(* CODESYS project PLS3 Flomsikring 28.07.2021.export

Project tree, tasks and I/O mapping:
  application PLS3_Flomsikring
    task MQTT (cyclic, interval 5000 ms, priority 15, watchdog 4500 ms x 1) calls Simulation_MQTT
    task PLC_Task (cyclic, interval 500 ms, priority 15, watchdog 400 ms x 1) calls PLC_PRG
    task VISU_TASK (cyclic, interval 100 ms, priority 15) calls VisuElems.Visu_Prg
    GlobalData/
      global variables HMI
      global variables IO
      global variables Local
      global variables SIM
      global variables STATUS
    LibFB/
      function block AlarmDigitalFB [ST]
      function block ControlAnalogFB [ST]
      function block MotorDigitalFB [ST]
      function block PIDFB [ST]
      function block PowerMonitoringFb [ST]
      function block ScalingFB [ST]
      function block SignalAnalogFB [ST]
      function block signalDigitalFB [ST]
      function block TimerFB [ST]
      function block WorkDistributorFB [ST]
    LibHmiStructs/
      data type AlarmDigitalHmiCmd
      data type AlarmDigitalHmiPv
      data type AliveHmiPv
      data type ControlAnalogHmiCmd
      data type ControlAnalogHmiPv
      data type MotorDigitalHmiCmd
      data type MotorDigitalHmiPv
      data type PIDHmiCmd
      data type PIDHmiPv
      data type PowerMonitoringHmiCmd
      data type PowerMonitoringHmiPv
      data type ScalingHmiCmd
      data type ScalingHmiPv
      data type SignalAnalogHmiCmd
      data type SignalAnalogHmiPv
      data type SignalDigitalHmiCmd
      data type SignalDigitalHmiPv
      data type TimerHmiCmd
      data type TimerHmiPv
      data type WorkDistributorHmiPv
    Utils/
      data type OpcUa_Mqtt_Status
      function eulers [ST]
      function firstOrderSystem [ST]
      function process [ST]
      function String_To_ForcastArray [ST]
    program Alarms [ST]
    program Control [ST]
    program Initialize [ST]
    program Inputs [ST]
    program Outputs [ST]
    program PLC_PRG [ST]
    function RestartOpcUaMqttLinkOnDownload [ST]
    function RestartOpcUaMqttLinkOnOnlineChange [ST]
    program Simulation [ST]
    program Simulation_MQTT [ST]
    global variables PersistentVars
    visualisation Visualization
*)

// PLS3_Flomsikring/LibHmiStructs/AlarmDigitalHmiCmd
// These are autogenerated, do not manual modify it
TYPE AlarmDigitalHmiCmd :
STRUCT
	_tagId: STRING;
	_type: STRING;
	_owner: STRING;
	Tag:	STRING;
	Description:	STRING;
	Delay:	TimerHmiCmd;
	Acknowledged:	BOOL;
END_STRUCT
END_TYPE

// PLS3_Flomsikring/LibHmiStructs/AlarmDigitalHmiPv
// These are autogenerated, do not manual modify it
TYPE AlarmDigitalHmiPv :
STRUCT
	_tagId: STRING;
	_type: STRING;
	_owner: STRING;
	Input_Pv:	BOOL;
	Delay:	TimerHmiPv;
	Alarm:	BOOL;
END_STRUCT
END_TYPE

// PLS3_Flomsikring/LibHmiStructs/AliveHmiPv
// These are autogenerated, do not manual modify it
TYPE AliveHmiPv :
STRUCT
	_tagId:STRING;
	_type: STRING;
	_owner: STRING;
	CounterPv:INT;
END_STRUCT
END_TYPE

// PLS3_Flomsikring/LibHmiStructs/ControlAnalogHmiCmd
// These are autogenerated, do not manual modify it
TYPE ControlAnalogHmiCmd :
STRUCT
	_tagId: STRING;
	_type: STRING;
	_owner: STRING;
	Tag:STRING;
	Description:STRING;
	Auto:BOOL;
	ManualControlValue_Cmd:REAL;
	AlarmControlFailed:	AlarmDigitalHmiCmd;
	AlarmControlFailedLimit:	REAL;
END_STRUCT
END_TYPE

// PLS3_Flomsikring/LibHmiStructs/ControlAnalogHmiPv
// These are autogenerated, do not manual modify it
TYPE ControlAnalogHmiPv :
STRUCT
	_tagId: STRING;
	_type: STRING;
	_owner: STRING;
	ControlValue_Pv:	REAL;
	Interlocked_Pv:	BOOL;
	AlarmControlFailed:	AlarmDigitalHmiPv;
	Feedback_Pv:REAL;
	RunHours_Pv:INT;
	RunMinutes_Pv:int;
END_STRUCT
END_TYPE

// PLS3_Flomsikring/LibHmiStructs/MotorDigitalHmiCmd
// These are autogenerated, do not manual modify it
TYPE MotorDigitalHmiCmd :
STRUCT
_tagId: STRING;
_type: STRING;
_owner: STRING;
Tag:STRING;
Description:STRING;
Auto:BOOL;
AlarmStartFailed:AlarmDigitalHmiCmd;
AlarmStopFailed:AlarmDigitalHmiCmd;
ManualStart_Cmd:BOOL;
END_STRUCT
END_TYPE

// PLS3_Flomsikring/LibHmiStructs/MotorDigitalHmiPv
// These are autogenerated, do not manual modify it
TYPE MotorDigitalHmiPv :
STRUCT
_tagId: STRING;
_type: STRING;
_owner: STRING;
Interlocked_Pv:BOOL;
ControlValue_Pv:BOOL;
AlarmStartFailed:AlarmDigitalHmiPv;
AlarmStopFailed:AlarmDigitalHmiPv;
Started_Pv:BOOL;
Stopped_Pv:BOOL;
END_STRUCT
END_TYPE

// PLS3_Flomsikring/LibHmiStructs/PIDHmiCmd
// These are autogenerated, do not manual modify it
TYPE PIDHmiCmd :
STRUCT
	_tagId: STRING;
	_type: STRING;
	_owner: STRING;
	Tag:STRING;
	Description:STRING;
	K:REAL;
	EnableK:BOOL;
	Ti:REAL;
	EnableI:BOOL;
	Td:REAL;
	N:REAL;
	EnableD:BOOL;
	Auto:BOOL;
	ManualValue_Cmd:REAL;
	u0:REAL;
	TrackingGain:REAL;
	HmiReference_Cmd:REAL;
	HmiReference:BOOL;
END_STRUCT
END_TYPE

// PLS3_Flomsikring/LibHmiStructs/PIDHmiPv
// These are autogenerated, do not manual modify it
TYPE PIDHmiPv :
STRUCT
	_tagId: STRING;
	_type: STRING;
	_owner: STRING;
	Reference_Pv:REAL;
	ProcessMeasure:REAL;
	Error:REAL;
	Output:REAL;
	up:REAL;
	ui:REAL;
	ud:REAL;
	es:REAL;
	u:REAL;
END_STRUCT
END_TYPE

// PLS3_Flomsikring/LibHmiStructs/PowerMonitoringHmiCmd
//These are autogenerated, do not manual modify it
TYPE PowerMonitoringHmiCmd :
STRUCT
	_tagId: STRING;
	_type: STRING;
	_owner: STRING;
	BatterySize_Cmd:REAL; //Size of the battery in mAh
END_STRUCT
END_TYPE

// PLS3_Flomsikring/LibHmiStructs/PowerMonitoringHmiPv
//These are autogenerated, do not manual modify it
TYPE PowerMonitoringHmiPv :
STRUCT
_tagId: STRING;
_type: STRING;
_owner: STRING;
Status_string:STRING;
Status_bool:BOOL;
Time_string:STRING;
Time_pv:REAL;
Alarm:BOOL;
Input_Current_In:REAL;
Input_Current_Out:REAL;
Input_Battery_Level:REAL;
END_STRUCT
END_TYPE

// PLS3_Flomsikring/LibHmiStructs/ScalingHmiCmd
// These are autogenerated, do not manual modify it
TYPE ScalingHmiCmd :
STRUCT
	_tagId: STRING;
	_type: STRING;
	_owner: STRING;
	InputUnit:STRING;
	InputMin_Cmd:REAL;
	InputMax_Cmd:REAL;
	OutputUnit:STRING;
	OutputMin_Cmd:REAL;
	OutputMax_Cmd:REAL;
END_STRUCT
END_TYPE

// PLS3_Flomsikring/LibHmiStructs/ScalingHmiPv
// These are autogenerated, do not manual modify it
TYPE ScalingHmiPv :
STRUCT
_tagId: STRING;
_type: STRING;
_owner: STRING;
Input_Pv:REAL;
Output_Pv:REAL;
END_STRUCT
END_TYPE

// PLS3_Flomsikring/LibHmiStructs/SignalAnalogHmiCmd
// These are autogenerated, do not manual modify it
TYPE SignalAnalogHmiCmd :
STRUCT
_tagId: STRING;
_type: STRING;
_owner: STRING;
Tag:STRING;
Description:STRING;
AlarmHigh:AlarmDigitalHmiCmd;
AlarmHighHigh:AlarmDigitalHmiCmd;
AlarmLow:AlarmDigitalHmiCmd;
AlarmLowLow:AlarmDigitalHmiCmd;
AlarmHighLimit:REAL;
AlarmHighHighLimit:REAL;
AlarmLowLimit:REAL;
AlarmLowLowLimit:REAL;
AlarmHysteresis:REAL;
SimulationMode:BOOL;
SimulationValue:REAL;
InputScaling:ScalingHmiCmd;
END_STRUCT
END_TYPE

// PLS3_Flomsikring/LibHmiStructs/SignalAnalogHmiPv
// These are autogenerated, do not manual modify it
TYPE SignalAnalogHmiPv :
STRUCT
_tagId: STRING;
_type: STRING;
_owner: STRING;
RawInput_Pv:REAL;
Output_Pv:REAL;
AlarmHigh:AlarmDigitalHmiPv;
AlarmHighHigh:AlarmDigitalHmiPv;
AlarmLow:AlarmDigitalHmiPv;
AlarmLowLow:AlarmDigitalHmiPv;
InputScaling:ScalingHmiPv;
END_STRUCT
END_TYPE

// PLS3_Flomsikring/LibHmiStructs/SignalDigitalHmiCmd
// These are autogenerated, do not manual modify it
TYPE SignalDigitalHmiCmd :
STRUCT
_tagId: STRING;
_type: STRING;
_owner: STRING;
Tag:STRING;
Description:STRING;
SimulationMode:BOOL;
SimulationValue:BOOL;
END_STRUCT
END_TYPE

// PLS3_Flomsikring/LibHmiStructs/SignalDigitalHmiPv
// These are autogenerated, do not manual modify it
TYPE SignalDigitalHmiPv :
STRUCT
_tagId: STRING;
_type: STRING;
_owner: STRING;
Input_Pv:BOOL;
Output_Pv:BOOL;
END_STRUCT
END_TYPE

// PLS3_Flomsikring/LibHmiStructs/TimerHmiCmd
// These are autogenerated, do not manual modify it
TYPE TimerHmiCmd :
STRUCT
	_tagId:STRING;
	_type: STRING;
	_owner: STRING;
	Tag:	STRING;
	Description:	STRING;
	OnDelayLimit:	REAL;
	OffDelayLimit:	REAL;
END_STRUCT
END_TYPE

// PLS3_Flomsikring/LibHmiStructs/TimerHmiPv
// These are autogenerated, do not manual modify it
TYPE TimerHmiPv :
STRUCT
	_tagId:STRING;
	_type: STRING;
	_owner: STRING;
	Input_Pv:	BOOL;
	Output_Pv:	BOOL;
	OnDelayElapsed:	REAL;
	OffDelayElapsed:	REAL;
END_STRUCT
END_TYPE

// PLS3_Flomsikring/LibHmiStructs/WorkDistributorHmiPv
// These are autogenerated, do not manual modify it
TYPE WorkDistributorHmiPv :
STRUCT
_tagId:STRING;
_type:STRING;
_owner:STRING;
Tag1:STRING;
Tag2:STRING;
Tag3:STRING;
RunHours1:INT;
RunHours2:INT;
RunHours3:INT;
AlarmNotAuto:BOOL;
END_STRUCT
END_TYPE

// PLS3_Flomsikring/Utils/OpcUa_Mqtt_Status
TYPE OpcUa_Mqtt_Status :
STRUCT
	LastRun:STRING;
	AliveCounterPv:INT := 0;
	Restart_Cmd:BOOL := FALSE;
END_STRUCT
END_TYPE

// PLS3_Flomsikring/PersistentVars
{attribute 'qualified_only'}
VAR_GLOBAL PERSISTENT RETAIN

	// Generated instance path of persistent variable
	HMI.AliveCounterPlc3Pv: AliveHmiPv;
	// Generated instance path of persistent variable
	HMI.ValveEmission1Cmd: ControlAnalogHmiCmd;
	// Generated instance path of persistent variable
	HMI.ValveEmission1Pv: ControlAnalogHmiPv;
	// Generated instance path of persistent variable
	HMI.ValveEmission1AlarmMotorProtectionCmd: AlarmDigitalHmiCmd;
	// Generated instance path of persistent variable
	HMI.ValveEmission1AlarmMotorProtectionPv: AlarmDigitalHmiPv;
	// Generated instance path of persistent variable
	HMI.ValveEmission1SignalDigitalMotorProtectionCmd: SignalDigitalHmiCmd;
	// Generated instance path of persistent variable
	HMI.ValveEmission1SignalDigitalMotorProtectionPv: SignalDigitalHmiPv;
	// Generated instance path of persistent variable
	HMI.ValveEmission1ScalingPositionCmd: ScalingHmiCmd;
	// Generated instance path of persistent variable
	HMI.ValveEmission1ScalingPositionPv: ScalingHmiPv;
	// Generated instance path of persistent variable
	HMI.ValveEmission1ScalingControlValueCmd: ScalingHmiCmd;
	// Generated instance path of persistent variable
	HMI.ValveEmission1ScalingControlValuePv: ScalingHmiPv;
	// Generated instance path of persistent variable
	HMI.ValveEmission1PIDCmd: PIDHmiCmd;
	// Generated instance path of persistent variable
	HMI.ValveEmission1PIDPv: PIDHmiPv;
	// Generated instance path of persistent variable
	HMI.WaterLevelCmd: SignalAnalogHmiCmd;
	// Generated instance path of persistent variable
	HMI.WaterLevelPv: SignalAnalogHmiPv;
	// Generated instance path of persistent variable
	HMI.FlowLevelEmissionCmd: SignalAnalogHmiCmd;
	// Generated instance path of persistent variable
	HMI.FlowLevelEmissionPv: SignalAnalogHmiPv;
END_VAR

// PLS3_Flomsikring/GlobalData/HMI
{attribute 'qualified_only'}
VAR_GLOBAL PERSISTENT RETAIN
	AliveCounterPlc3Pv:AliveHmiPv;
	ValveEmission1Cmd: ControlAnalogHmiCmd;
	ValveEmission1Pv: ControlAnalogHmiPv;
	ValveEmission1AlarmMotorProtectionCmd:AlarmDigitalHmiCmd;
	ValveEmission1AlarmMotorProtectionPv:AlarmDigitalHmiPv;
	ValveEmission1SignalDigitalMotorProtectionCmd:SignalDigitalHmiCmd;
	ValveEmission1SignalDigitalMotorProtectionPv:SignalDigitalHmiPv;
	ValveEmission1ScalingPositionCmd:ScalingHmiCmd;
	ValveEmission1ScalingPositionPv:ScalingHmiPv;
	ValveEmission1ScalingControlValueCmd:ScalingHmiCmd;
	ValveEmission1ScalingControlValuePv:ScalingHmiPv;
	ValveEmission1PIDCmd: PIDHmiCmd;
	ValveEmission1PIDPv: PIDHmiPv;
	
	WaterLevelCmd: SignalAnalogHmiCmd;
	WaterLevelPv: SignalAnalogHmiPv;
	
	FlowLevelEmissionCmd: SignalAnalogHmiCmd;
	FlowLevelEmissionPv: SignalAnalogHmiPv;

END_VAR

// PLS3_Flomsikring/GlobalData/IO
{attribute 'qualified_only'}
VAR_GLOBAL
	DI_ValveEmission1MotorProtectionOk: BOOL := TRUE;
	
	AI_ValveEmission1PositionPv:REAL;
	AI_WaterLevelPv:REAL;
	AI_FlowLevelEmmissionPv:REAL;
	
	AO_ValveEmission1ControlValue:REAL;
END_VAR

// PLS3_Flomsikring/GlobalData/Local
{attribute 'qualified_only'}
VAR_GLOBAL
	ValveEmission1:ControlAnalogFB;
	ValveEmission1PID:PIDFB;
	ValveEmission1AlarmMotorProtection:AlarmDigitalFB;
	ValveEmission1MotorProtectionOk:signalDigitalFB;
	ValveEmission1ScalingPosition:ScalingFB;
	ValveEmission1ScalingControlValue:ScalingFB;
	
	WaterLevel:SignalAnalogFB;
	FlowLevelEmission:SignalAnalogFB;
	
	RainForcast: ARRAY[0..4] OF REAL;
END_VAR

// PLS3_Flomsikring/GlobalData/SIM
{attribute 'qualified_only'}
VAR_GLOBAL
	WaterLevel_Pv_m:REAL;
	EmissionFlow_Pv_m3_s:REAL;
	ValveEmission1Position_Pv:REAL;
	RainForcast_m_day: ARRAY[0..4] OF REAL;
END_VAR

// PLS3_Flomsikring/GlobalData/STATUS
{attribute 'qualified_only'}
VAR_GLOBAL
	OpcUaMqttLinkStatus: OpcUa_Mqtt_Status;
END_VAR

// PLS3_Flomsikring/Simulation_MQTT
PROGRAM Simulation_MQTT
VAR
	MqttStatus 				: WagoAppCloud.FbStatus_NativeMQTT;
	MqttError				: BOOL := FALSE;
	MqttConnectedToMyCloud	: BOOL := FALSE;
	MqttFillLevel			: REAL := 0;
	MqttOutgoingBlocks		: ULINT := 0;
	
	
	
	MqttSubscribe 				: WagoAppCloud.FbSubscribeMQTT;
	MqttSubscriptionDataBytes	: ARRAY [0..254] OF BYTE;
	MqttSubscriptionDataJSONString			: STRING(JSON_MAX_STRING);	//	Resulting JSON string
	MqttSubscriptionDataJSONPointer			: WagoAppJSON.typJSON_Pointer;
	MqttSubcriptionJSONParser				: Fb_JSON_ParseAndModify;	//	JSON parser function block
	MqttSubscribeNewData: BOOL;
	
	oParserStatus	: WagoAppJSON.WagoSysErrorBase.FbResult;
	xParserError	: BOOL;
	xParserDone		: BOOL;
	diParserToken	: DINT;
	xParserBuildup	: BOOL;
	xParserTrigger	: ARRAY[0..5] OF BOOL;
	
	MqttPublish 		: WagoAppCloud.FbPublishMQTT;
	MqttPublishParameters	: ARRAY[0..10] OF STRING;
	MqttPublishTemplate		: STRING(512) := '{"#Parameter": #Parameter}';
	JSONWriter 		: FB_JSON_Writer_01;
	MqttPublishPayload		: STRING(1024);
	MqttPublishBuffer			: ARRAY[0..1999] OF BYTE;
	MqttPublishTrigger : BOOL;
	JSONWriter_Done	: BOOL;
	JSONWriter_Error	: BOOL;
	JSONWriter_Status		: WagoSysErrorBase.FbResult;
	JSONWriterTrigger	: BOOL;
END_VAR

// Status
MqttStatus(xEnabled := TRUE,
		   xError => MqttError,
		   xCloudConnected => MqttConnectedToMyCloud,			// Will be FALSE after network timeout occured 
		   rCacheFillLevel => MqttFillLevel,					// Increasing value indicates bad network or overload
		   uliOutgoingDataBlocks => MqttOutgoingBlocks);  	// Only for QoS 1 and 2. Increasing value indicates bad network or overload
		   
// Subscribe to data		   
MqttSubscribe(xSubscribe := TRUE, 
	sTopic := 'ba/wago/sim/plc3/plcsub', 
	eQoS := eQualityOfService.QoS1, 
	aPayloadData:= MqttSubscriptionDataBytes,
	xDataReceived => MqttSubscribeNewData);

MemCopySecure(pDest:= ADR(MqttSubscriptionDataJSONString), udiDestSize:= 255, pSource:= ADR(MqttSubscriptionDataBytes), udiSourceSize:= MqttSubscribe.dwRxNBytes, bPadding:= 0);

//	Execute this function block once to complete the parser buildup process
//	This must be done before calling the parser methods

IF MqttSubscribeNewData THEN
	xParserBuildup := TRUE;
END_IF

MqttSubcriptionJSONParser(
	pData:= ADR(MqttSubscriptionDataJSONString), 			//	JSON string to parse
	udiSizeData:= length(MqttSubscriptionDataJSONString), 
	oStatus=> oParserStatus, 
	xError=> xParserError, 
	xDone=> xParserDone, 
	diToken=> diParserToken, 
	xTrigger:= xParserBuildup);		//	Set xParserBuildup TRUE to execute the function block
	
IF xParserDone THEN
	xParserTrigger[0] := TRUE;			//	Set xParserTrigger TRUE to execute the parser method
	xParserTrigger[1] := TRUE;			
	xParserTrigger[2] := TRUE;			
	xParserTrigger[3] := TRUE;			
	xParserDone := FALSE;
END_IF

//	Call the parser method GetValueByPath for each value to be extracted from the JSON string
MqttSubscriptionDataJSONPointer := MqttSubcriptionJSONParser.GetValueByPath(sPointer:='/WaterLevel_Pv',xTrigger:=xParserTrigger[0]);
SIM.WaterLevel_Pv_m := STRING_TO_REAL(MqttSubscriptionDataJSONPointer.sValue);
MqttSubscriptionDataJSONPointer := MqttSubcriptionJSONParser.GetValueByPath(sPointer:='/EmissionFlow_Pv',xTrigger:=xParserTrigger[1]);
SIM.EmissionFlow_Pv_m3_s := STRING_TO_REAL(MqttSubscriptionDataJSONPointer.sValue);
MqttSubscriptionDataJSONPointer := MqttSubcriptionJSONParser.GetValueByPath(sPointer:='/RainForcast',xTrigger:=xParserTrigger[2]);
SIM.RainForcast_m_day := String_To_ForcastArray(MqttSubscriptionDataJSONPointer.sValue);

// Publish data
MqttPublishParameters[0] := 'ValveEmission1Position_Pv'; 
MqttPublishParameters[1] := REAL_TO_STRING(SIM.ValveEmission1Position_Pv);

JSONWriterTrigger := TRUE; // Parses every time this routine executes
JSONWriter(
	sJSON_BaseFrame:= MqttPublishTemplate, 
	oStatus=> JSONWriter_Status, 
	xError=> JSONWriter_Error, 
	xDone=> JSONWriter_Done, 
	aParameterValues:= MqttPublishParameters, 
	xTrigger:= JSONWriterTrigger, 
	sOutput:= MqttPublishPayload);

MemCopy(pDest := ADR(MqttPublishBuffer), pSource := ADR(MqttPublishPayload), udiSize := Length(MqttPublishPayload));

MqttPublishTrigger := TRUE; // Parses every time this routine executes
MqttPublish(sTopic := 'ba/wago/sim/plc3/plcpub',
			eQualityOfService := 1,
			dwSize :=  Length(MqttPublishPayload),
			aData := MqttPublishBuffer,
			xTrigger := MqttPublishTrigger);

END_PROGRAM

// PLS3_Flomsikring/Utils/process
FUNCTION process : REAL
VAR_INPUT
	u:REAL;
	Ts:REAL;
	y:REAL;
	yMin:REAL;
	yMax:REAL;
	T:REAL;
	Kp:REAL;
END_VAR
VAR
	_out:real;
END_VAR

_out := eulers(y, firstOrderSystem(T, Kp, y, u), Ts);
IF _out > yMax THEN
	_out := yMax;
ELSIF _out < yMin THEN
	_out := yMin;
END_IF;
process := _out;

END_FUNCTION

// PLS3_Flomsikring/Utils/eulers
FUNCTION eulers : REAL
VAR_INPUT
	y:REAL;
	f:REAL;
	h:REAL;
END_VAR
VAR
END_VAR

eulers := y + (h*f);

END_FUNCTION

// PLS3_Flomsikring/Utils/firstOrderSystem
FUNCTION firstOrderSystem : REAL
VAR_INPUT
	T:REAL;
	Kp:REAL;
	y:REAL;
	u:REAL;
END_VAR
VAR
END_VAR

firstOrderSystem :=  -(y/T) + ((Kp/T)*u);

END_FUNCTION

// PLS3_Flomsikring/Utils/String_To_ForcastArray
FUNCTION String_To_ForcastArray : ARRAY[0..4] OF REAL
VAR_INPUT
	InputString:STRING;
END_VAR
VAR
	temp:STRING;
	temp1:STRING;
	temp2:STRING;
	pos:INT;
	i:INT;
	values :ARRAY[0..4] OF REAL;
END_VAR

i := 0;

pos := LEN(InputString);
temp := DELETE(InputString, 1, 1);
temp1 := temp;
temp := DELETE(temp, 1, pos-1);
temp2 := temp;
pos := FIND(temp, ',');
FOR i := 0 TO 3 BY 1 DO
	values[i] := STRING_TO_REAL(LEFT(temp, pos-1)); // Denne tar ikke hensyn til siste verdi, då den leter etter komma men det finnes ikke
	temp := DELETE(temp, pos+2, 0);
	pos := FIND(temp, ',');
END_FOR;
values[4] := STRING_TO_REAL(temp);
String_To_ForcastArray := values;

END_FUNCTION

// PLS3_Flomsikring/PLC_PRG
PROGRAM PLC_PRG
VAR
	_firstScan:BOOL := TRUE;
	_counter:INT;
	_lastRun:STRING;
END_VAR



// Signaling that the PLC is alive
Hmi.AliveCounterPlc3Pv._tagId := 'AliveCounterPlc3Pv';
Hmi.AliveCounterPlc3Pv._type := 'AliveHmi';
Hmi.AliveCounterPlc3Pv._owner := 'plc3';
HMI.AliveCounterPlc3Pv.CounterPv := HMI.AliveCounterPlc3Pv.CounterPv + 1;


_counter := STATUS.OpcUaMqttLinkStatus.AliveCounterPv;
_lastRun := STATUS.OpcUaMqttLinkStatus.LastRun;

IF _firstScan THEN
	Initialize();
END_IF
Inputs();
Alarms();
Control();
Outputs();
Simulation();





// Always last
_firstScan := FALSE;

END_PROGRAM

// PLS3_Flomsikring/Initialize
PROGRAM Initialize
VAR
END_VAR


// First run setpoints - are stored while power failure, but not for program updates
Hmi.ValveEmission1SignalDigitalMotorProtectionCmd.Tag := 'VE01';
Hmi.ValveEmission1SignalDigitalMotorProtectionCmd.Description := 'Digital signal for Emission Valve 1 motor protection';

Hmi.ValveEmission1ScalingPositionCmd.InputMax_Cmd := 100.0;
Hmi.ValveEmission1ScalingPositionCmd.InputMin_Cmd := 0.0;
Hmi.ValveEmission1ScalingPositionCmd.OutputMax_Cmd := 100.0;
Hmi.ValveEmission1ScalingPositionCmd.OutputMin_Cmd := 0.0;

Hmi.ValveEmission1ScalingControlValueCmd.InputMax_Cmd := 100.0;
Hmi.ValveEmission1ScalingControlValueCmd.InputMin_Cmd := 0.0;
Hmi.ValveEmission1ScalingControlValueCmd.OutputMax_Cmd := 100.0;
Hmi.ValveEmission1ScalingControlValueCmd.OutputMin_Cmd := 0.0;

Hmi.ValveEmission1AlarmMotorProtectionCmd.Tag := 'VE01';
Hmi.ValveEmission1AlarmMotorProtectionCmd.Description := 'Motor protection alarm Emission Valve 1';
Hmi.ValveEmission1AlarmMotorProtectionCmd.Delay.OnDelayLimit := 1.0;
Hmi.ValveEmission1AlarmMotorProtectionCmd.Delay.OffDelayLimit := 5.0; 

HMI.ValveEmission1Cmd.Tag := 'VE01';
HMI.ValveEmission1Cmd.Description := 'Emission valve 1';
HMI.ValveEmission1Cmd.Auto := TRUE;
HMI.ValveEmission1Cmd.ManualControlValue_Cmd := 50.0;
HMI.ValveEmission1Cmd.AlarmControlFailedLimit := 10.0;
HMI.ValveEmission1Cmd.AlarmControlFailed.Description := 'Failed to control Emission valve 1';
HMI.ValveEmission1Cmd.AlarmControlFailed.Delay.OnDelayLimit := 100.0;
HMI.ValveEmission1Cmd.AlarmControlFailed.Delay.OffDelayLimit := 10.0;
HMI.ValveEmission1Cmd.AlarmControlFailed.Acknowledged := TRUE;

Hmi.ValveEmission1PIDCmd.Tag := 'PID02';
Hmi.ValveEmission1PIDCmd.Description := 'Regulator for controling emission valve 1';
Hmi.ValveEmission1PIDCmd.HmiReference := FALSE;
Hmi.ValveEmission1PIDCmd.HmiReference_Cmd := 20.0;
Hmi.ValveEmission1PIDCmd.Auto := TRUE;
Hmi.ValveEmission1PIDCmd.EnableK := TRUE;
Hmi.ValveEmission1PIDCmd.EnableI := TRUE;
Hmi.ValveEmission1PIDCmd.EnableD := FALSE;
Hmi.ValveEmission1PIDCmd.K := -207.0;
Hmi.ValveEmission1PIDCmd.Ti := 30.0;
Hmi.ValveEmission1PIDCmd.Td := 0.0;
Hmi.ValveEmission1PIDCmd.N := 10.0;
Hmi.ValveEmission1PIDCmd.TrackingGain := 1.0;
Hmi.ValveEmission1PIDCmd.u0 := 50.0;
Hmi.WaterLevelCmd.Tag := 'PT01';
Hmi.WaterLevelCmd.Description := 'Level of supply water';
Hmi.WaterLevelCmd.AlarmHysteresis := 1.0;
Hmi.WaterLevelCmd.AlarmHighHighLimit := 25.0;
Hmi.WaterLevelCmd.AlarmHighLimit := 24.5;
Hmi.WaterLevelCmd.AlarmLowLowLimit := 0.0;
Hmi.WaterLevelCmd.AlarmLowLimit := 0.0;
Hmi.WaterLevelCmd.AlarmHigh.Description := 'High level supply water';
Hmi.WaterLevelCmd.AlarmHigh.Delay.OnDelayLimit := 1.0;
Hmi.WaterLevelCmd.AlarmHigh.Delay.OffDelayLimit := 1.0;
Hmi.WaterLevelCmd.AlarmHighHigh.Description := 'High high level supply water';
Hmi.WaterLevelCmd.AlarmHighHigh.Delay.OnDelayLimit := 1.0;
Hmi.WaterLevelCmd.AlarmHighHigh.Delay.OffDelayLimit := 1.0;
Hmi.WaterLevelCmd.AlarmLow.Description := 'Low level supply water';
Hmi.WaterLevelCmd.AlarmLow.Delay.OnDelayLimit := 1.0;
Hmi.WaterLevelCmd.AlarmLow.Delay.OffDelayLimit := 1.0;
Hmi.WaterLevelCmd.AlarmLowLow.Description := 'Low low level supply water';
Hmi.WaterLevelCmd.AlarmLowLow.Delay.OnDelayLimit := 1.0;
Hmi.WaterLevelCmd.AlarmLowLow.Delay.OffDelayLimit := 1.0;
Hmi.WaterLevelCmd.InputScaling.InputUnit := 'na';
Hmi.WaterLevelCmd.InputScaling.OutputUnit := 'm';
Hmi.WaterLevelCmd.InputScaling.InputMax_Cmd := 100.0;
Hmi.WaterLevelCmd.InputScaling.InputMin_Cmd := 0.0;
Hmi.WaterLevelCmd.InputScaling.OutputMax_Cmd := 100.0;
Hmi.WaterLevelCmd.InputScaling.OutputMin_Cmd := 0.0;

Hmi.FlowLevelEmissionCmd.Tag := 'FT08';
Hmi.FlowLevelEmissionCmd.Description := 'Level of flow out of water';
Hmi.FlowLevelEmissionCmd.AlarmHysteresis := 3.0;
Hmi.FlowLevelEmissionCmd.AlarmHighHighLimit := 900.0;
Hmi.FlowLevelEmissionCmd.AlarmHighLimit := 800.0;
Hmi.FlowLevelEmissionCmd.AlarmLowLowLimit := 0.0;
Hmi.FlowLevelEmissionCmd.AlarmLowLimit := 0.0;
Hmi.FlowLevelEmissionCmd.AlarmHigh.Delay.OnDelayLimit := 1.0;
Hmi.FlowLevelEmissionCmd.AlarmHigh.Delay.OffDelayLimit := 1.0;
Hmi.FlowLevelEmissionCmd.AlarmHighHigh.Delay.OnDelayLimit := 1.0;
Hmi.FlowLevelEmissionCmd.AlarmHighHigh.Delay.OffDelayLimit := 1.0;
Hmi.FlowLevelEmissionCmd.AlarmLow.Delay.OnDelayLimit := 1.0;
Hmi.FlowLevelEmissionCmd.AlarmLow.Delay.OffDelayLimit := 1.0;
Hmi.FlowLevelEmissionCmd.AlarmLowLow.Delay.OnDelayLimit := 1.0;
Hmi.FlowLevelEmissionCmd.AlarmLowLow.Delay.OffDelayLimit := 1.0;
Hmi.FlowLevelEmissionCmd.AlarmHighHigh.Description := 'HighHigh emission flow';
Hmi.FlowLevelEmissionCmd.AlarmHigh.Description := 'High emission flow';
Hmi.FlowLevelEmissionCmd.AlarmLow.Description := 'Low emission flow';
Hmi.FlowLevelEmissionCmd.AlarmLowLow.Description := 'Low low emission flow';
Hmi.FlowLevelEmissionCmd.InputScaling.InputUnit := 'na';
Hmi.FlowLevelEmissionCmd.InputScaling.OutputUnit := 'l/s';
Hmi.FlowLevelEmissionCmd.InputScaling.InputMax_Cmd := 100.0;
Hmi.FlowLevelEmissionCmd.InputScaling.InputMin_Cmd := 0.0;
Hmi.FlowLevelEmissionCmd.InputScaling.OutputMax_Cmd := 100.0;
Hmi.FlowLevelEmissionCmd.InputScaling.OutputMin_Cmd := 0.0;

END_PROGRAM

// PLS3_Flomsikring/Control
PROGRAM Control
VAR
	_reference_default_m: REAL := 22.0;
	_reference_m: REAL;
END_VAR

// Adjusting setpoint to prevent to much water in the river

_reference_m := _reference_default_m - Local.RainForcast[2];


// Regulator block
Local.ValveEmission1PID(_id := 'ValveEmission1PID', _owner := 'plc3',
	InputReference := _reference_m,
	ProcessMeasure := Local.WaterLevel.Output,
	Ts := 0.5,
	uMax := 100.0,
	uMin := 0.0,
	HmiCmd := Hmi.ValveEmission1PIDCmd,
	HmiPv := Hmi.ValveEmission1PIDPv);

	

// Valves
Local.ValveEmission1(_id := 'ValveEmission1', _owner := 'plc3',
	HmiCmd := HMI.ValveEmission1Cmd,
	HmiPv := HMI.ValveEmission1Pv,
	Interlock := NOT Local.ValveEmission1MotorProtectionOk.Output,
	Feedback := Local.ValveEmission1ScalingPosition.Output,
	ControlValueAuto_Cmd := Local.ValveEmission1PID.Output); // ControlValueAuto_Cmd from PID regulator

END_PROGRAM

// PLS3_Flomsikring/Inputs
PROGRAM Inputs
VAR
	
END_VAR



Local.ValveEmission1MotorProtectionOk(_id := 'ValveEmission1SignalDigitalMotorProtection', _owner := 'plc3',
									Input := IO.DI_ValveEmission1MotorProtectionOk,
									HmiCmd := HMI.ValveEmission1SignalDigitalMotorProtectionCmd,
									HmiPv := HMI.ValveEmission1SignalDigitalMotorProtectionPv);

// We dont need the scaling, but a real system would
Local.ValveEmission1ScalingPosition(_id := 'ValveEmission1ScalingPosition', _owner := 'plc3',
						Input := IO.AI_ValveEmission1PositionPv,
						HmiCmd := HMI.ValveEmission1ScalingPositionCmd,
						HmiPv := HMI.ValveEmission1ScalingPositionPv);


Local.WaterLevel(_id := 'WaterLevel', _owner := 'plc3',
				RawInput := IO.AI_WaterLevelPv,
				HmiCmd := HMI.WaterLevelCmd,
				HmiPv := HMI.WaterLevelPv);
				
Local.FlowLevelEmission(_id := 'FlowLevelEmission', _owner := 'plc3',
				RawInput := IO.AI_FlowLevelEmmissionPv,
				HmiCmd := HMI.FlowLevelEmissionCmd,
				HmiPv := HMI.FlowLevelEmissionPv);

END_PROGRAM

// PLS3_Flomsikring/Alarms
PROGRAM Alarms
VAR
END_VAR



Local.ValveEmission1AlarmMotorProtection(_id := 'ValveEmission1AlarmMotorProtection', _owner := 'plc3',
										HmiCmd := HMI.ValveEmission1AlarmMotorProtectionCmd,
										HmiPv := HMI.ValveEmission1AlarmMotorProtectionPv,
										Input := NOT Local.ValveEmission1MotorProtectionOk.Output);

END_PROGRAM

// PLS3_Flomsikring/Outputs
PROGRAM Outputs
VAR
END_VAR


// We dont need the scaling, but a real system would
Local.ValveEmission1ScalingControlValue(_id := 'ValveEmission1ScalingControlValue', _owner := 'plc3',
						Input := Local.ValveEmission1.ControlValue,
						HmiCmd := HMI.ValveEmission1ScalingControlValueCmd,
						HmiPv := HMI.ValveEmission1ScalingControlValuePv,
						Output => IO.AO_ValveEmission1ControlValue);

END_PROGRAM

// PLS3_Flomsikring/Simulation
PROGRAM Simulation
VAR
END_VAR

// Simulation because we need to be able to change the forcast to fit our need
Local.RainForcast := SIM.RainForcast_m_day;

// Simulation because no physical IO is connected

IO.DI_ValveEmission1MotorProtectionOk := True;
// Simulating valve follows controlvalue
//IO.AI_ValveEmission1PositionPv := IO.AO_ValveEmission1ControlValue; // TODO add first order delay function


IO.AI_ValveEmission1PositionPv := process(u := IO.AO_ValveEmission1ControlValue,
	Ts := 0.5, y := IO.AI_ValveEmission1PositionPv, yMin := 0.001, yMax := 100.0, T := 2.0,  Kp := 1.0);

SIM.ValveEmission1Position_Pv := IO.AI_ValveEmission1PositionPv;
IO.AI_WaterLevelPv := SIM.WaterLevel_Pv_m;
IO.AI_FlowLevelEmmissionPv := SIM.EmissionFlow_Pv_m3_s;

END_PROGRAM

// PLS3_Flomsikring/RestartOpcUaMqttLinkOnDownload
FUNCTION RestartOpcUaMqttLinkOnDownload : DWORD
VAR_IN_OUT
	EventPrm: CmpApp.EVTPARAM_CmpApp;
END_VAR
VAR
END_VAR

(*
This function is called whan a download is about to happen. 
This will force the Opc Ua - MQTT link to restart.
The restart will take 10 seconds, allowing e!Cockpit to download and start before the link starts.
*)
Status.OpcUaMqttLinkStatus.Restart_Cmd := TRUE;

END_FUNCTION

// PLS3_Flomsikring/RestartOpcUaMqttLinkOnOnlineChange
FUNCTION RestartOpcUaMqttLinkOnOnlineChange : DWORD
VAR_IN_OUT
	EventPrm: CmpApp.EVTPARAM_CmpApp;
END_VAR
VAR
END_VAR

(*
This function is called whan a online change is about to happen. 
This will force the Opc Ua - MQTT link to restart.
The restart will take 10 seconds, allowing e!Cockpit to download and start before the link starts.
*)
Status.OpcUaMqttLinkStatus.Restart_Cmd := TRUE;

END_FUNCTION

// PLS3_Flomsikring/LibFB/AlarmDigitalFB
FUNCTION_BLOCK AlarmDigitalFB
VAR_INPUT
	_id:STRING;
	_owner:STRING;
	Input:	BOOL;
END_VAR
VAR_OUTPUT
	Alarm:	BOOL;
END_VAR
VAR
	_Delay:	TimerFB;
	_AlarmLastScan:BOOL;
	_type:string := 'AlarmDigital';
END_VAR
VAR_IN_OUT
	HmiCmd:	AlarmDigitalHmiCmd;
	HmiPv:	AlarmDigitalHmiPv;
END_VAR

(*
Name: AlarmDigitalFB
Author: Jone Vassbø
Version: 0.3
Date: 09.03.2020
Description:
- Function block for a digital alarm, with commands from HMI in seperate struct
*)

// In routine - start -
// Validate input
// In routine - end -
// Alarm routine - start
// Alarm routine - end -

// Control routine - start -
_Delay(_id := _id, _owner := _owner, Input := Input, Output => Alarm, HmiCmd := HmiCmd.Delay, HmiPv := HmiPv.Delay);
IF Alarm AND NOT _AlarmLastScan THEN // Flank
	HmiCmd.Acknowledged := FALSE;
END_IF
_AlarmLastScan := Alarm;
// Control routine - end -

// Out routine - start - 
HmiPv.Input_Pv := Input;
HmiPv.Alarm := Alarm OR NOT HmiCmd.Acknowledged;
HmiCmd._tagId := CONCAT(_id, 'Cmd');
HmiPv._tagId := CONCAT(_id, 'Pv');
HmiPv._type := _type;
HmiCmd._type := _type;
HmiPv._owner := _owner;
HmiCmd._owner := _owner;
// Out routine - end -

END_FUNCTION_BLOCK

// PLS3_Flomsikring/LibFB/TimerFB
FUNCTION_BLOCK TimerFB
VAR_INPUT
	_id:STRING;
	_owner:STRING;
	Input:	BOOL;
END_VAR
VAR_OUTPUT
	Output:	BOOL;
END_VAR
VAR
	OnDelay: TON;
	OffDelay: TOF;
	ToSec:REAL := 1000.0;
	_type:string := 'Timer';
END_VAR
VAR_IN_OUT
	HmiCmd:	TimerHmiCmd;
	HmiPv: TimerHmiPv;
END_VAR

(*
Name: TimerFB
Author: Jone Vassbø
Version: 0.4
Date: 09.03.2020
Description:
- Function block operating as a Timer with both on and off delay
*)

// In routine - start -
// Validate input
IF HmiCmd.OnDelayLimit < 0 THEN
	HmiCmd.OnDelayLimit := 0.0;
END_IF
IF HmiCmd.OffDelayLimit < 0 THEN
	HmiCmd.OnDelayLimit := 0.0;
END_IF
// In routine - end -
// Alarm routine - start
// Alarm routine - end -
// Control routine - start -
OnDelay(IN := Input,
	PT := TO_TIME(HmiCmd.OnDelayLimit*ToSec));
HmiPv.OnDelayElapsed := TO_REAL(OnDelay.ET)/ToSec;

OffDelay(IN := OnDelay.Q,
	PT := TO_TIME(HmiCmd.OffDelayLimit*ToSec));
HmiPv.OffDelayElapsed := TO_REAL(OffDelay.ET)/ToSec;

IF OnDelay.Q THEN
	Output := TRUE;
END_IF
IF NOT OffDelay.Q THEN
	Output := FALSE;
END_IF
// Control routine - end -

// Out routine - start - 
HmiPv.Input_Pv := Input;
HmiPv.Output_Pv := Output;
HmiCmd._tagId := CONCAT(_id, 'Cmd');
HmiPv._tagId := CONCAT(_id, 'Pv');
HmiPv._type := _type;
HmiCmd._type := _type;
HmiPv._owner := _owner;
HmiCmd._owner := _owner;
// Out routine - end -

END_FUNCTION_BLOCK

// PLS3_Flomsikring/LibFB/ControlAnalogFB
FUNCTION_BLOCK ControlAnalogFB
VAR_INPUT
	_id:STRING;
	_owner:STRING;
	ControlValueAuto_Cmd:REAL;
	Interlock:BOOL;
	Feedback:REAL;
END_VAR
VAR_OUTPUT
	ControlValue:REAL;
	Alarm:BOOL;
END_VAR
VAR
	_AlarmControlFailed: AlarmDigitalFB;
	_hoursTimer:TON;
	_type:STRING := 'ControlAnalog';
END_VAR
VAR_IN_OUT
	HmiCmd:	ControlAnalogHmiCmd;
	HmiPv:	ControlAnalogHmiPv;
END_VAR

(*
Name: ValveAnalogFB
Author: Jone Vassbø
Version: 0.3
Date: 09.03.2020
Description:
- Function block to control a analog valve, with commands from HMI in seperate struct
*)

// In routine - start -
// Validate input
IF HmiCmd.ManualControlValue_Cmd > 100.0 THEN
	HmiCmd.ManualControlValue_Cmd := 100.0;
END_IF
IF HmiCmd.ManualControlValue_Cmd < 0.0 THEN
	HmiCmd.ManualControlValue_Cmd := 0.0;
END_IF
IF ControlValueAuto_Cmd > 100.0 THEN
	ControlValueAuto_Cmd := 100.0;
END_IF
IF ControlValueAuto_Cmd < 0.0 THEN
	ControlValueAuto_Cmd := 0.0;
END_IF
// In routine - end -
// Alarm routine - start
_AlarmControlFailed(_id := _id, _owner := _owner, Input := ABS(Feedback - ControlValue) > HmiCmd.AlarmControlFailedLimit,
	HmiCmd := HmiCmd.AlarmControlFailed, HmiPv := HmiPv.AlarmControlFailed);
// Alarm routine - end -

// Control routine - start -
IF Interlock OR Alarm THEN
	HmiCmd.Auto := FALSE;
	HmiCmd.ManualControlValue_Cmd := 0.0;
END_IF

IF HmiCmd.auto THEN
	ControlValue := ControlValueAuto_Cmd;
ELSE
	ControlValue := HmiCmd.ManualControlValue_Cmd;
END_IF

_hoursTimer(In:= (ControlValue > 0.3) AND NOT _hoursTimer.Q, PT:= T#0.0416666667S);
// Using HmiPv because the tag is retain
IF _hoursTimer.Q THEN
	HmiPv.RunMinutes_Pv := HmiPv.RunMinutes_Pv + 1; 
END_IF
IF HmiPv.RunMinutes_Pv = 60 THEN
	HmiPv.RunHours_Pv := HmiPv.RunHours_Pv + 1;
	HmiPv.RunMinutes_Pv := 0;
END_IF
IF HmiPv.RunHours_Pv < 0 THEN
	HmiPv.RunHours_Pv := 0;
END_IF

// Control routine - end -

// Out routine - start - 
Alarm := _AlarmControlFailed.Alarm OR NOT HmiCmd.AlarmControlFailed.Acknowledged;
HmiPv.ControlValue_Pv := ControlValue;
HmiPv.Interlocked_Pv := Interlock;
HmiPv.Feedback_Pv := Feedback;
HmiCmd._tagId := CONCAT(_id, 'Cmd');
HmiPv._tagId := CONCAT(_id, 'Pv');
HmiPv._type := _type;
HmiCmd._type := _type;
HmiPv._owner := _owner;
HmiCmd._owner := _owner;
// Out routine - end -

END_FUNCTION_BLOCK

// PLS3_Flomsikring/LibFB/MotorDigitalFB
FUNCTION_BLOCK MotorDigitalFB
VAR_INPUT
	_id:STRING;
	_owner:STRING;
	Interlock:BOOL;
	ControlValueAuto_Cmd:BOOL;
	Started:BOOL;
	Stopped:BOOL;
END_VAR
VAR_OUTPUT
	ControlValue:BOOL;
	Alarm:BOOL;
END_VAR
VAR
	_StartFailed:AlarmDigitalFB;
	_StopFailed:AlarmDigitalFB;
	_type:string := 'MotorDigital';
END_VAR
VAR_IN_OUT
	HmiCmd:MotorDigitalHmiCmd;
	HmiPv:MotorDigitalHmiPv;
END_VAR

(*
Name: MotorDigitalFB
Author: Jone Vassbø
Version: 0.3
Date: 09.03.2020
Description:
- Function block to control a digital motor, with commands from HMI in seperate struct
*)

// In routine - start -
// Validate input
// In routine - end -
// Alarm routine - start
_StartFailed(_id := _id, _owner := _owner, Input := (NOT Started AND ControlValue) OR (Started AND NOT ControlValue),
	HmiCmd := HmiCmd.AlarmStartFailed, HmiPv := HmiPv.AlarmStartFailed);
_StopFailed(_id := _id, _owner := _owner, Input := (Stopped AND ControlValue) OR (NOT Stopped AND NOT ControlValue),
	HmiCmd := HmiCmd.AlarmStopFailed, HmiPv := HmiPv.AlarmStopFailed);
// Alarm routine - end -

// Control routine - start -
IF Interlock OR Alarm THEN
	HmiCmd.auto := FALSE;
	HmiCmd.ManualStart_Cmd := FALSE;
END_IF

IF HmiCmd.auto THEN
	ControlValue := ControlValueAuto_Cmd;
ELSE
	ControlValue := HmiCmd.ManualStart_Cmd;
END_IF
// Control routine - end -

// Out routine - start - 
Alarm := _StartFailed.Alarm OR NOT HmiCmd.AlarmStartFailed.Acknowledged OR _StopFailed.Alarm OR NOT HmiCmd.AlarmStopFailed.Acknowledged;
HmiPv.ControlValue_Pv := ControlValue;
HmiPv.Interlocked_Pv := Interlock;
HmiPv.Started_Pv := Started;
HmiPv.Stopped_Pv := Stopped;
HmiCmd._tagId := CONCAT(_id, 'Cmd');
HmiPv._tagId := CONCAT(_id, 'Pv');
HmiPv._type := _type;
HmiCmd._type := _type;
HmiPv._owner := _owner;
HmiCmd._owner := _owner;
// Out routine - end -

END_FUNCTION_BLOCK

// PLS3_Flomsikring/LibFB/PIDFB
FUNCTION_BLOCK PIDFB
VAR_INPUT
	_id:STRING;
	_owner:STRING;
	InputReference:REAL;
	ProcessMeasure:REAL;
	Ts:REAL;
	uMax:REAL;
	uMin:REAL;
END_VAR
VAR_OUTPUT
	Output:REAL;
	Out_e:REAL;
	Out_up:REAL;
	Out_ui:REAL;
	Out_ud:REAL;
	Out_es:REAL;
	Out_u:REAL;
END_VAR
VAR
	_type:STRING := 'PID';
	
	y_last:REAL := 0.0;
	u_limited:REAL := 0.0;
	u:REAL := 0.0;
	e:REAL := 0.0;
	es:REAL := 0.0;
	manual_last:BOOL := FALSE;
	// P
	up:REAL := 0.0;
	// I
	alfa:REAL := 0.0;
	ui:REAL := 0.0;
	ui_last:REAL := 0.0;
	enableI_last:BOOL := TRUE;
	// D
	ud:REAL := 0.0;
	ud_last:REAL := 0.0;
	beta:REAL := 0.0;
	ref:REAL:= 0;
END_VAR
VAR_IN_OUT
	HmiCmd:PIDHmiCmd;
	HmiPv:PIDHmiPv;
END_VAR

(*
Name: PIDFB
Author: Jone Vassbø
Version: 0.1
Date: 09.03.2020
Description:
-  Standard PID regulatior block
*)

IF HmiCmd.HmiReference THEN
	ref := HmiCmd.HmiReference_Cmd;
ELSE
	ref := InputReference;
END_IF


e := ref - ProcessMeasure;
// K
up := (HmiCmd.K * e)*BOOL_TO_REAL(HmiCmd.EnableK);

// I
alfa := Ts / HmiCmd.Ti;
ui := (ui_last + (HmiCmd.K * alfa * e) + (es*(1/HmiCmd.TrackingGain)))*BOOL_TO_REAL(HmiCmd.EnableI);        
ui_last := ui;
// On enable I
IF HmiCmd.EnableI AND NOT enableI_last THEN
	ui := HmiCmd.u0;
END_IF;
// On disable I
IF NOT HmiCmd.EnableI AND enableI_last THEN
	HmiCmd.u0 := ui;
END_IF;

enableI_last := HmiCmd.enableI;
// D
beta := HmiCmd.Td / (HmiCmd.Td + (Ts * HmiCmd.N));
ud := ((beta * ud_last) - (HmiCmd.K * (HmiCmd.Td / Ts) * (1 - beta) * (ProcessMeasure - y_last))) * BOOL_TO_REAL(HmiCmd.enableD);
ud_last := ud;
y_last := ProcessMeasure;

u := HmiCmd.u0 + up + ui + ud;

// On enable manual
IF NOT HmiCmd.Auto AND NOT manual_last THEN
	HmiCmd.ManualValue_Cmd := u;
END_IF;
IF NOT HmiCmd.Auto THEN
	u_limited := HmiCmd.ManualValue_Cmd;
ELSE
	u_limited := u;
END_IF;
IF u_limited > uMax THEN
	u_limited := uMax;
ELSIF u_limited < uMin THEN
	u_limited := uMin;
END_IF;

manual_last := NOT HmiCmd.Auto;
es := u_limited - u;

Output := u_limited;
Out_e := e;
Out_up := up;
Out_ui := ui;
Out_ud := ud;
Out_es := es;
Out_u := u;

HmiPv.Reference_Pv := ref;
HmiPv.ProcessMeasure := ProcessMeasure;
HmiPv.Error := e;
HmiPv.Output := Output;
HmiPv.up := up;
HmiPv.ui := ui;
HmiPv.ud := ud;
HmiPv.es := es;
HmiPv.u := u;

HmiCmd._tagId := CONCAT(_id, 'Cmd');
HmiPv._tagId := CONCAT(_id, 'Pv');
HmiPv._type := _type;
HmiCmd._type := _type;
HmiPv._owner := _owner;
HmiCmd._owner := _owner;

END_FUNCTION_BLOCK

// PLS3_Flomsikring/LibFB/PowerMonitoringFb
FUNCTION_BLOCK PowerMonitoringFb
VAR_INPUT
	_id:STRING;
	_owner:STRING;
	Input_CurrentIn:REAL;
	Input_CurrentOut:REAL;
	Input_CurrentStored:REAL;
END_VAR
VAR_OUTPUT
END_VAR
VAR
	_type:STRING:= 'PowerMonitoring';
	Current_balance :REAL;
END_VAR
VAR_IN_OUT
	HmiCmd:PowerMonitoringHmiCmd;
	HmiPv:PowerMonitoringHmiPv;
END_VAR

(*
Name: PowerMonitoringFB
Author: Markus Raudberget
Version: 0.1
Date: 14.03.2020
Description:
- Function block for Power monitoring of a battery package, with commands from hmi i seperate struct
*)

//Control routine - start -
Current_balance := (Input_currentIn - Input_CurrentOut);
IF Current_balance <0 THEN
	HmiPv.Status_bool :=FALSE;
	HmiPv.Status_string :='Decharging';
	HmiPv.Time_pv := Input_CurrentStored / -Current_balance;
	HmiPv.Time_string :='Time for empty battery';
ELSE 
	HmiPv.Status_bool :=TRUE;
	HmiPv.Status_string :='Charging';
	HmiPv.Time_pv := (HmiCmd.BatterySize_Cmd - Input_CurrentStored) / Current_balance;
	HmiPv.Time_string :='Time for full battery';
END_IF

HmiPv.Input_Current_In :=Input_CurrentIn;
HmiPv.Input_Current_Out :=Input_CurrentOut;
HmiPv.Input_Battery_Level :=Input_CurrentStored;

HmiCmd._tagId := CONCAT(_id, 'Cmd');
HmiPv._tagId := CONCAT(_id, 'Pv');
HmiPv._type := _type;
HmiCmd._type := _type;
HmiPv._owner := _owner;
HmiCmd._owner := _owner;

END_FUNCTION_BLOCK

// PLS3_Flomsikring/LibFB/ScalingFB
FUNCTION_BLOCK ScalingFB
VAR_INPUT
	_id:STRING;
	_owner:STRING;
	Input:REAL;
END_VAR
VAR_OUTPUT
	Output:REAL;
END_VAR
VAR
	_type:string := 'Scaling';
END_VAR
VAR_IN_OUT
	HmiCmd:ScalingHmiCmd;
	HmiPv:ScalingHmiPv;
END_VAR


(*
Name: ScalingFB
Author: Jone Vassbø
Version: 0.3
Date: 09.03.2020
Description:
- Function block for a scaling analog value, with commands from HMI in seperate struct
*)

// Control routine - start -
Output :=  HmiCmd.OutputMin_Cmd * (1 - ((Input - HmiCmd.InputMin_Cmd) / (HmiCmd.InputMax_Cmd - HmiCmd.InputMin_Cmd))) + HmiCmd.OutputMax_Cmd * ((Input - HmiCmd.InputMin_Cmd) / (HmiCmd.InputMax_Cmd - HmiCmd.InputMin_Cmd));
// Control routine - end -

// Out routine - start - 
HmiPv.Input_Pv := Input;
HmiPv.Output_Pv := Output;
HmiCmd._tagId := CONCAT(_id, 'Cmd');
HmiPv._tagId := CONCAT(_id, 'Pv');
HmiPv._type := _type;
HmiCmd._type := _type;
HmiCmd._owner := _owner;
HmiPv._owner := _owner;
// Out routine - end -

END_FUNCTION_BLOCK

// PLS3_Flomsikring/LibFB/SignalAnalogFB
FUNCTION_BLOCK SignalAnalogFB
VAR_INPUT
	_id:STRING;
	_owner:STRING;
	RawInput:REAL;
END_VAR
VAR_OUTPUT
	Output:REAL;
	AlarmHigh:BOOL;
	AlarmHighHigh:BOOL;
	AlarmLow:BOOL;
	AlarmLowLow:BOOL;
END_VAR
VAR
	_AlarmHigh: AlarmDigitalFB;
	_AlarmHighHigh: AlarmDigitalFB;
	_AlarmLow: AlarmDigitalFB;
	_AlarmLowLow: AlarmDigitalFB;
	_Scaling: ScalingFB;
	
	_High:BOOL;
	_HighHigh:BOOL;
	_Low:BOOL;
	_LowLow:BOOL;
	
	_type:string := 'SignalAnalog';
END_VAR
VAR_IN_OUT
	HmiCmd:SignalAnalogHmiCmd;
	HmiPv:SignalAnalogHmiPv;
END_VAR

(*
Name: SignalAnalogFB
Author: Jone Vassbø
Version: 0.3
Date: 09.03.2020
Description:
- Function block for a analog signal, with alarms and commands from HMI in seperate struct
*)

// In routine - start -
// Validate input
_Scaling(_id := _id, _owner := _owner, Input:= RawInput, HmiCmd := HmiCmd.InputScaling, HmiPv := HmiPv.InputScaling);
IF HmiCmd.SimulationMode THEN
	Output := HmiCmd.SimulationValue;
ELSE
	Output := _Scaling.Output;
END_IF
// In routine - end -
// Alarm routine - start
IF Output > HmiCmd.AlarmHighLimit THEN
	_High := TRUE;
END_IF
IF Output < (HmiCmd.AlarmHighLimit - HmiCmd.AlarmHysteresis) THEN
	_High := FALSE;
END_IF
_AlarmHigh(_id := _id, _owner := _owner, Input :=  _High,
	HmiCmd := HmiCmd.AlarmHigh, HmiPv := HmiPv.AlarmHigh);

IF Output > HmiCmd.AlarmHighHighLimit THEN
	_HighHigh := TRUE;
END_IF
IF Output < (HmiCmd.AlarmHighHighLimit - HmiCmd.AlarmHysteresis) THEN
	_HighHigh := FALSE;
END_IF
_AlarmHighHigh(_id := _id, _owner := _owner, Input :=  _HighHigh,
	HmiCmd := HmiCmd.AlarmHighHigh, HmiPv := HmiPv.AlarmHighHigh);

IF Output < HmiCmd.AlarmLowLimit THEN
	_Low := TRUE;
END_IF
IF Output > (HmiCmd.AlarmLowLimit + HmiCmd.AlarmHysteresis) THEN
	_Low := FALSE;
END_IF
_AlarmLow(_id := _id, _owner := _owner, Input :=  _Low,
	HmiCmd := HmiCmd.AlarmLow, HmiPv := HmiPv.AlarmLow);
	
IF Output < HmiCmd.AlarmLowLowLimit THEN
	_LowLow := TRUE;
END_IF
IF Output > (HmiCmd.AlarmLowLowLimit + HmiCmd.AlarmHysteresis) THEN
	_LowLow := FALSE;
END_IF
_AlarmLowLow(_id := _id, _owner := _owner, Input :=  _LowLow,
	HmiCmd := HmiCmd.AlarmLowLow, HmiPv := HmiPv.AlarmLowLow);
// Alarm routine - end -

// Control routine - start -

// Control routine - end -

// Out routine - start - 
AlarmHigh := _AlarmHigh.Alarm OR NOT HmiCmd.AlarmHigh.Acknowledged;
AlarmHighHigh := _AlarmHighHigh.Alarm OR NOT HmiCmd.AlarmHighHigh.Acknowledged;
AlarmLow := _AlarmLow.Alarm OR NOT HmiCmd.AlarmLow.Acknowledged;
AlarmLowLow := _AlarmLowLow.Alarm OR NOT HmiCmd.AlarmLowLow.Acknowledged;

HmiPv.Output_Pv := Output;
HmiPv.RawInput_Pv := RawInput;
HmiCmd._tagId := CONCAT(_id, 'Cmd');
HmiPv._tagId := CONCAT(_id, 'Pv');
HmiPv._type := _type;
HmiCmd._type := _type;
HmiPv._owner := _owner;
HmiCmd._owner := _owner;
// Out routine - end -

END_FUNCTION_BLOCK

// PLS3_Flomsikring/LibFB/signalDigitalFB
FUNCTION_BLOCK signalDigitalFB
VAR_INPUT
	_id:STRING;
	_owner:STRING;
	Input:BOOL;
END_VAR
VAR_OUTPUT
	Output:BOOL;
END_VAR
VAR
	_type:string := 'SignalDigital';
END_VAR
VAR_IN_OUT
	HmiCmd:SignalDigitalHmiCmd;
	HmiPv:SignalDigitalHmiPv;
END_VAR

(*
Name: signalDigitalFB
Author: Jone Vassbø
Version: 0.3
Date: 09.03.2020
Description:
- Function block for a digital signal, with commands from HMI in seperate struct
*)

// In routine - start -
// Validate input
// In routine - end -
// Alarm routine - start
// Alarm routine - end -

// Control routine - start -
IF HmiCmd.SimulationMode THEN
	Output := HmiCmd.SimulationValue;
ELSE
	Output := Input;
END_IF
// Control routine - end -

// Out routine - start - 
HmiPv.Input_Pv := Input;
HmiPv.Output_Pv := Output;
HmiCmd._tagId := CONCAT(_id, 'Cmd');
HmiPv._tagId := CONCAT(_id, 'Pv');
HmiPv._type := _type;
HmiCmd._type := _type;
HmiPv._owner := _owner;
HmiCmd._owner := _owner;
// Out routine - end -

END_FUNCTION_BLOCK

// PLS3_Flomsikring/LibFB/WorkDistributorFB
FUNCTION_BLOCK WorkDistributorFB
VAR_INPUT
	_id:STRING;
	_owner:STRING;
	InputControlSignal:REAL;
	Tag1:STRING;
	Tag2:STRING;
	Tag3:STRING;
	InAuto1:BOOL;
	InAuto2:BOOL;
	InAuto3:BOOL;
	RunHours1:INT;
	RunHours2:INT;
	RunHours3:INT;
	ChangeInterval:REAL;
END_VAR
VAR_OUTPUT
	Out1:REAL;
	Out2:REAL;
	Out3:REAL;

END_VAR
VAR
	_intervalTimer:TON;
	_alarm:BOOL;
	_type:STRING := 'WorkDistributor';
	_ToSec:REAL := 1000.0;
	_maxWorkingHours:INT;
	_run1:BOOL;
	_run2:BOOL;
	_run3:BOOL;
END_VAR
VAR_IN_OUT
	HmiPv:WorkDistributorHmiPv;
END_VAR

(*
Name: WorkDistributorFB
Author: Jone Vassbø
Version: 0.4
Date: 09.03.2020
Description:
- Function block to distribute work between three components
*)

_intervalTimer(IN := NOT _intervalTimer.Q,
	PT := TO_TIME(ChangeInterval*_ToSec));

_alarm := NOT InAuto1 OR NOT InAuto2 OR NOT InAuto3;

// These are located here because of the return statments
HmiPv.Tag1 := Tag1;
HmiPv.Tag2 := Tag2;
HmiPv.Tag3 := Tag3;
HmiPv.RunHours1 := RunHours1;
HmiPv.RunHours2 := RunHours2;
HmiPv.RunHours3 := RunHours3;
HmiPv.AlarmNotAuto := _alarm;

HmiPv._tagId := CONCAT(_id, 'Pv');
HmiPv._type := _type;
HmiPv._owner := _owner;

IF _alarm THEN
	Out1 := InputControlSignal;
	Out2 := InputControlSignal;
	Out3 := InputControlSignal;
	RETURN;
END_IF

Out1 := (InputControlSignal*BOOL_TO_REAL(_run1)); 
Out2 := (InputControlSignal*BOOL_TO_REAL(_run2));
Out3 := (InputControlSignal*BOOL_TO_REAL(_run3));


// Time to change who is working
IF _intervalTimer.Q THEN
	_run1 := TRUE;
	_run2 := TRUE;
	_run3 := TRUE;
	
	_maxWorkingHours := RunHours1;
	IF RunHours2 > _maxWorkingHours THEN
		_maxWorkingHours := RunHours2;
	END_IF
	IF RunHours3 > _maxWorkingHours THEN
		_maxWorkingHours := RunHours3;
	END_IF

	IF RunHours1 = _maxWorkingHours THEN
		_run1 := FALSE;
		RETURN; // Prevents two from stopping
	END_IF
	IF RunHours2 = _maxWorkingHours THEN
		_run2 := FALSE;
		RETURN;
	END_IF
	IF RunHours3 = _maxWorkingHours THEN
		_run3 := FALSE;
		RETURN;
	END_IF
END_IF

END_FUNCTION_BLOCK

// PLS3_Flomsikring/Visualization
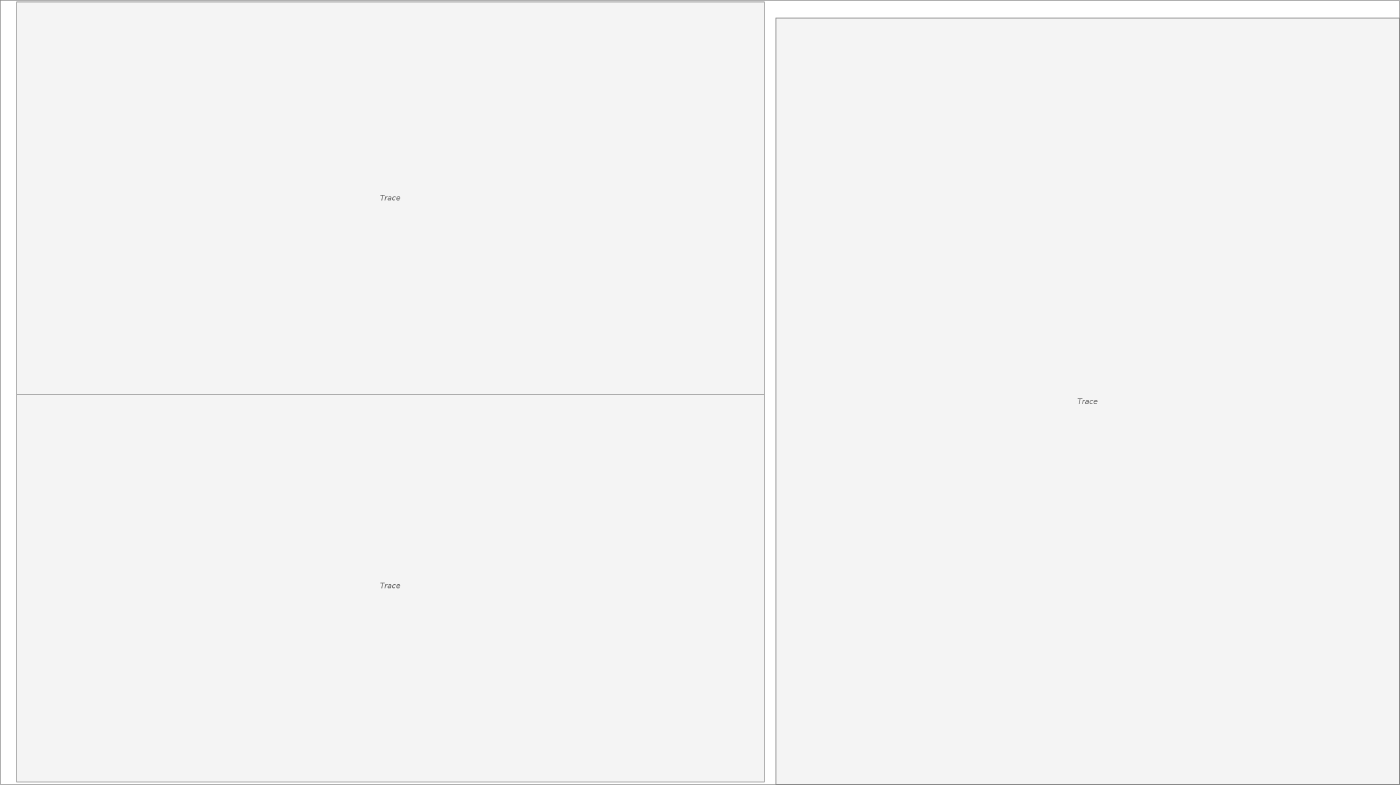
VISUALIZATION Visualization  // 1892x1061
    Trace (22,526 1011x531)
    Trace (1048,24 844x1037)
    Trace (22,2 1011x531)
END_VISUALIZATION
